// Mitsubishi GX Works2 project: SmartFarmModbusTemp01   PLC: FX3U/FX3UC

PROGRAM MAIN
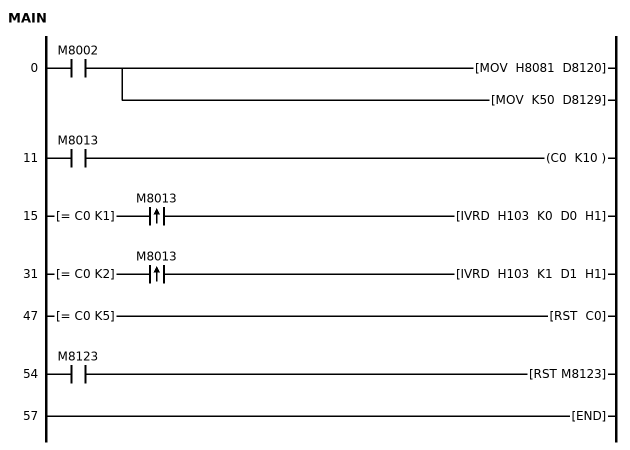
0     LD      M8002
      MOV     H8081 D8120
      MOV     K50 D8129
11    LD      M8013
      OUT     C0 K10
15    LD=     C0 K1
      ANDP    M8013
      IVRD    H103 K0 D0 H1
31    LD=     C0 K2
      ANDP    M8013
      IVRD    H103 K1 D1 H1
47    LD=     C0 K5
      RST     C0
54    LD      M8123
      RST     M8123
57    END
END_PROGRAM
